% RSLogix 500 project JEFF TEST PANEL_BAK008.RSS, saved by version 11.00.00.00 %
PROJECT "ML1400"    % processor: MicroLogix 1400; MAIN_PROG %

PROGRAM FILES
  LAD 2 "MAIN_PROG"  4 rungs

DATA FILES
  O0 OUTPUT  6 elements
  I1 INPUT  8 elements
  S2 STATUS  66 elements
  B3 BINARY  1 elements
  T4 TIMER  3 elements
  C5 COUNTER  1 elements
  R6 CONTROL  1 elements
  N7 INTEGER  3 elements
  F8 FLOAT  1 elements

LADDER 2 "MAIN_PROG"
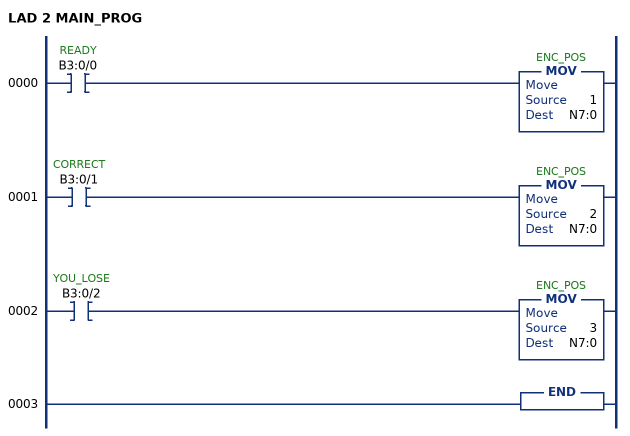
% Rung: 0 %
SOR XIC B3:0/0 MOV 1 N7:0 EOR
%   B3:0/0  READY %
%   N7:0  ENC_POS %
% Rung: 1 %
SOR XIC B3:0/1 MOV 2 N7:0 EOR
%   B3:0/1  CORRECT %
%   N7:0  ENC_POS %
% Rung: 2 %
SOR XIC B3:0/2 MOV 3 N7:0 EOR
%   B3:0/2  YOU_LOSE %
%   N7:0  ENC_POS %
% Rung: 3 %
SOR END EOR

OTHER DOCUMENTED ADDRESSES
  I:0.0/0  ENC_BIT0
  I:0.0/1  ENC_BIT1
  I:0.0/2  ENC_BIT2
  I:0.0/3  ENC_BIT3
  I:0.0/4  ENC_BIT4
  I:0.0/5  ENC_BIT5
  I:0.0/6  ENC_BIT6
  I:0.0/7  ENC_BIT7
  N7:0/1  "DEC2"
  N7:0/2  "DEC4"
  N7:0/3  "DEC8"
  N7:0/4  "DEC16"
  N7:0/5  "DEC32"
  N7:0/6  "DEC64"
  N7:0/7  "DEC128"
  N7:1  HMI
  N7:2  CRADDLE_DOWN_POSITIO
  T4:0  TIMER_ON_DELAY
  T4:1  TIMER_OFF_DELAY
  T4:2  RETENTITIVE_ON_DEALY

COMMENTS NOT ATTACHED TO A CURRENT RUNG
  N7:0/7: Read all 8 bits of the Encoder and convert to Gray Code
  N7:2: Subtract 76 from the gray code to find the absolute position

DATA TABLE (non-zero values as saved)
DATA B3
% B3:0 % 0X0001
DATA T4
% .PRE .ACC %
% T4:0 % 10 10
% T4:1 % 10 10
% T4:2 % 10 0
DATA N7
% N7:0 % 229 0 153
